{attribute 'GeneratedUsingTerminal: EJ1100-0000-0018'}
{attribute addProperty BoxType "EJ1100-0000-0018"}
{attribute addProperty Description "EJ1100 EtherCAT Coupler (2.2A E-Bus)"}
{attribute addProperty Physics "YKY"}
{attribute addProperty Id "InfoDataAT %I*InfoData_6F19DB2B2"}
{attribute addProperty CRC "532711307"}
{attribute addProperty Size "2"}
TYPE EJ1100_1FC0878B EXTENDS EtcSlaveBoxBase_77A0E4A7 :
STRUCT
	{attribute addProperty Name "InfoData"}
	InfoData : InfoData_6F19DB2B;
END_STRUCT
END_TYPE
